{attribute wpf [Container(Layout.Stack)]}
FUNCTION_BLOCK Station001_Components EXTENDS TcoCore.TcoObject
VAR	
	{attribute addProperty Name "Horizontal axis"}
	_horizontalAxis : DriveSim(THIS^);
	{attribute addProperty Name "Vertical piston"}
	_verticalPiston : TcoPneumatics.TcoCylinder(THIS^);
	{attribute addProperty Name "Gripper piston"}
	_gripperPiston : TcoPneumatics.TcoCylinder(THIS^);
END_VAR
VAR
	_counter : ULINT;
	_simulationCycle : BOOL;
END_VAR

_counter := _counter + 1;
_simulationCycle := (_counter MOD 500) = 0;


IF(IO.qA1[0] AND _simulationCycle) THEN
	IO.iA1[0] := TRUE;
	IO.iA1[1] := FALSE;
END_IF

IF(IO.qA1[1] AND _simulationCycle) THEN
	IO.iA1[1] := TRUE;
	IO.iA1[0] := FALSE;
END_IF

_verticalPiston(inoAtHomePos:= IO.iA1[0], inoAtWorkPos:= IO.iA1[1], inoToHomePos:= IO.qA1[0], inoToWorkPos:=IO.qA1[1] );


IF(IO.qA1[2] AND _simulationCycle) THEN
	IO.iA1[2] := TRUE;
	IO.iA1[3] := FALSE;
END_IF

IF(IO.qA1[3] AND _simulationCycle) THEN
	IO.iA1[3] := TRUE;
	IO.iA1[2] := FALSE;
END_IF

_gripperPiston(inoAtHomePos:= IO.iA1[2], inoAtWorkPos:= IO.iA1[3], inoToHomePos:= IO.qA1[2], inoToWorkPos:=IO.qA1[3]);


_horizontalAxis();

PROPERTY Gripper :  REFERENCE TO TcoPneumatics.TcoCylinder
GET
Gripper REF= _gripperPiston;
END_GET
END_PROPERTY

PROPERTY HorizontalAxis : IDrive
GET
HorizontalAxis := _horizontalAxis;
END_GET
END_PROPERTY

METHOD Service : BOOL
VAR_INPUT
END_VAR
_horizontalAxis.Service();
_verticalPiston.Service();
_gripperPiston.Service();
END_METHOD

PROPERTY VerticalAxis : REFERENCE TO TcoPneumatics.TcoCylinder
GET
VerticalAxis REF= _verticalPiston;
END_GET
END_PROPERTY

END_FUNCTION_BLOCK

(* stored: Version 1.1.0.1, ProductVersion 3.1.4024.9
   POU Station001_Components: Id {e806c847-ecc4-43b0-a026-69e0b11f80ef}, SpecialFunc None
   Property Gripper: Id {45058c8f-3b79-49b6-8729-6389402fa4b0}
   Get Get: Id {d387ff5f-f5d6-44a8-b450-cb493513cbfe}
   Property HorizontalAxis: Id {b1ab433f-e84d-4bd1-b49e-16adbd28465d}
   Get Get: Id {7f862521-62c1-4810-98b0-73ca60cc7784}
   Method Service: Id {98457207-8a91-45fe-bd57-5bb0d15033a9}
   Property VerticalAxis: Id {95519e2e-c8d9-4542-adf0-78464b1acba5}
   Get Get: Id {2a859788-f8eb-4b2b-8a8a-19eb876b8488} *)
